PROGRAM PB_Initialisation
VAR
    Initialised : BOOL;
    OnlineChangeCount : UDINT := 999;
END_VAR

IF NOT Initialised OR _AppInfo.OnlineChangeCnt <> OnlineChangeCount THEN
    // Re-link notification handlers...
    LinkNotificationHandlers();
    Initialised := TRUE;
    OnlineChangeCount := _AppInfo.OnlineChangeCnt;
END_IF

METHOD LinkNotificationHandlers
Objects.Safety.EStopTripped
    .ClearNotificationHandlers()
    .AddNotificationHandler(Objects.Machine.NotificationHandler_OnEstopTripped)
    .AddNotificationHandler(Objects.HydraulicPumpMotor.NotificationHandler_OnEstopTripped);

Objects.Safety.EStopReset
    .ClearNotificationHandlers()
    .AddNotificationHandler(Objects.Machine.NotificationHandler_OnEstopReset)
    .AddNotificationHandler(Objects.HydraulicPumpMotor.NotificationHandler_OnEstopReset);

// Notifications declared in the base class library, raised by all instances of T_Execution  
tcl_BaseClasses.GlobalEvents.Notification_ExecutionAborted
    .ClearNotificationHandlers()
    .AddNotificationHandler(Objects.Logging.NotificationHandler_OnExecutionAborted);

tcl_BaseClasses.GlobalEvents.Notification_ExecutionFailed
    .ClearNotificationHandlers()
    .AddNotificationHandler(Objects.Logging.NotificationHandler_OnExecutionFailed);

// Notification handlers accessed via properties...    
Notifications.Notification_OnUserLoggedIn
    .ClearNotificationHandlers()
    .AddNotificationHandler(Objects.Logging.NotificationHandler_OnUserLoggedIn);

Notifications.Notification_OnUserLoggedOut
    .ClearNotificationHandlers()
    .AddNotificationHandler(Objects.Logging.NotificationHandler_OnUserLoggedOut);
END_METHOD

END_PROGRAM

(* stored: Version 1.1.0.1, ProductVersion 3.1.4024.9
   POU PB_Initialisation: Id {fb4d6021-4d29-42c6-9db1-7c12735a2aa1}, SpecialFunc None
   Method LinkNotificationHandlers: Id {fe8ec0cd-8985-0afe-11e4-c25169e5a51e} *)
